{attribute addProperty BoxType "EL2521-0124-0016"}
{attribute addProperty Id "PLS_EnabledAT %I*BOOL811Status_of_outputAT %I*BOOL814Sync_ErrorAT %I*BOOL8132TxPDO_ToggleAT %I*BOOL819"}
{attribute addProperty CRC "2969786769"}
{attribute addProperty SizeInBites "32"}
{attribute addProperty SizeInBytes "4"}
TYPE PLS_Status_B1035991 :
STRUCT
	{attribute addProperty Name "PLS_Enabled"}
	PLS_Enabled AT %I* : BOOL;
	{attribute addProperty Name "Status_of_output"}
	Status_of_output AT %I* : BOOL;
	{attribute addProperty Name "Sync_Error"}
	Sync_Error AT %I* : BOOL;
	{attribute addProperty Name "TxPDO_Toggle"}
	TxPDO_Toggle AT %I* : BOOL;
END_STRUCT
END_TYPE

(* stored: Version 1.2.0.0, ProductVersion 3.1.4024.9
   DUT PLS_Status_B1035991: Id {c3b78b48-e7e7-4a6c-a15b-6c688a28cb4d} *)
